FUNCTION_BLOCK FB_Escort_monitoring
VAR_INPUT
	Coil_Lh1:BOOL;
	Coil_Lh2:BOOL;
	Coil_Rh1:BOOL;
	Coil_Rh2:BOOL;
	Valve_Lh1_open:BOOL;
	Valve_Lh1_closed:BOOL;
	Valve_Lh2_open:BOOL;
	Valve_Lh2_closed:BOOL;
	Valve_Rh1_open:BOOL;
	Valve_Rh1_closed:BOOL;
	Valve_Rh2_open:BOOL;
	Valve_Rh2_closed:BOOL;
	Open_time:TIME;
	Close_time:TIME;
END_VAR
VAR_OUTPUT
	Lh1_not_opening:BOOL;
	Lh1_not_closing:BOOL;
	Lh1_open_and_closed:BOOL;
	Lh2_not_opening:BOOL;
	Lh2_not_closing:BOOL;
	Lh2_open_and_closed:BOOL;
	Rh1_not_opening:BOOL;
	Rh1_not_closing:BOOL;
	Rh1_open_and_closed:BOOL;
	Rh2_not_opening:BOOL;
	Rh2_not_closing:BOOL;
	Rh2_open_and_closed:BOOL;
	Lh1_with_brakes_on:BOOL;
	Lh2_with_brakes_on:BOOL;
	Rh1_with_brakes_on:BOOL;
	Rh2_with_brakes_on:BOOL;
	Lh1_Lh2_xcheck:BOOL;
	Rh1_Rh2_xcheck:BOOL;
	Lh1_chatter:BOOL;
	Lh2_chatter:BOOL;
	Rh1_chatter:BOOL;
	Rh2_chatter:BOOL;
END_VAR
VAR
	Reset_chatter_counters:BOOL;
	FB_Valve_monitor_0: FB_Valve_monitor;
	FB_Valve_monitor_1: FB_Valve_monitor;
	FB_Valve_monitor_2: FB_Valve_monitor;
	FB_Valve_monitor_3: FB_Valve_monitor;
	TON_0: TON;
	TON_1: TON;
	TON_2: TON;
	TON_3: TON;
	R_TRIG_0: R_TRIG;
	CTU_0: CTU;
	CTU_1: CTU;
	CTU_2: CTU;
	CTU_3: CTU;
END_VAR

Escort_valves();

METHOD Escort_valves
VAR_INPUT
END_VAR
{warning "TODO: Address %S7 needs to be correctly addressed}
VAR_INST // added by the converter: edge detectors and wires of the graphical bodies
    _w1, _w5 : ANY;
    _w2, _w3, _w4 : BOOL;
END_VAR
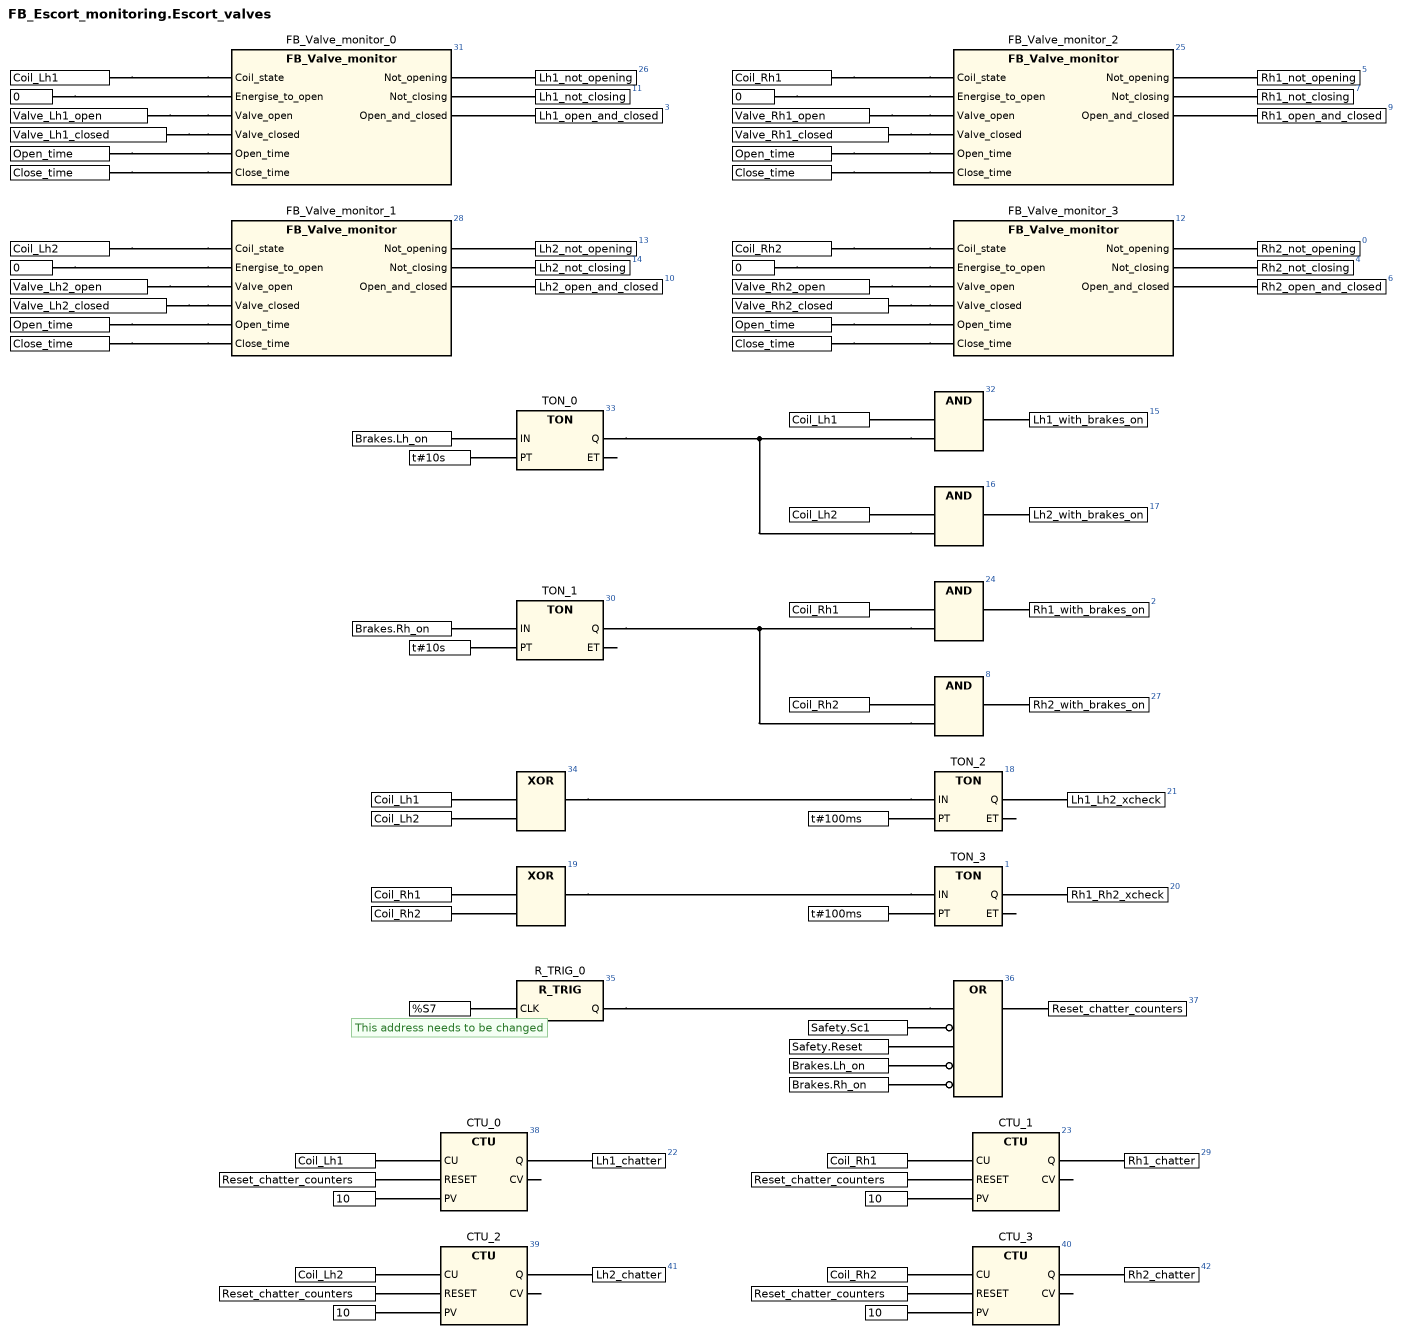
Rh2_not_opening := FB_Valve_monitor_3.Not_opening;
TON_3(IN := _w1, PT := t#100ms); // TON
Rh1_with_brakes_on := _w2;
Lh1_open_and_closed := FB_Valve_monitor_0.Open_and_closed;
Rh2_not_closing := FB_Valve_monitor_3.Not_closing;
Rh1_not_opening := FB_Valve_monitor_2.Not_opening;
Rh2_open_and_closed := FB_Valve_monitor_3.Open_and_closed;
Rh1_not_closing := FB_Valve_monitor_2.Not_closing;
_w3 := Coil_Rh2 AND TON_1.Q;
Rh1_open_and_closed := FB_Valve_monitor_2.Open_and_closed;
Lh2_open_and_closed := FB_Valve_monitor_1.Open_and_closed;
Lh1_not_closing := FB_Valve_monitor_0.Not_closing;
FB_Valve_monitor_3(
    Coil_state := Coil_Rh2,
    Energise_to_open := 0,
    Valve_open := Valve_Rh2_open,
    Valve_closed := Valve_Rh2_closed,
    Open_time := Open_time,
    Close_time := Close_time); // FB_Valve_monitor
Lh2_not_opening := FB_Valve_monitor_1.Not_opening;
Lh2_not_closing := FB_Valve_monitor_1.Not_closing;
Lh1_with_brakes_on := _w4;
Lh2_with_brakes_on := Coil_Lh2 AND TON_0.Q;
TON_2(IN := _w5, PT := t#100ms); // TON
_w1 := Coil_Rh1 XOR Coil_Rh2;
Rh1_Rh2_xcheck := TON_3.Q;
Lh1_Lh2_xcheck := TON_2.Q;
Lh1_chatter := CTU_0.Q;
CTU_1(CU := Coil_Rh1, RESET := Reset_chatter_counters, PV := 10); // CTU
_w2 := Coil_Rh1 AND TON_1.Q;
FB_Valve_monitor_2(
    Coil_state := Coil_Rh1,
    Energise_to_open := 0,
    Valve_open := Valve_Rh1_open,
    Valve_closed := Valve_Rh1_closed,
    Open_time := Open_time,
    Close_time := Close_time); // FB_Valve_monitor
Lh1_not_opening := FB_Valve_monitor_0.Not_opening;
Rh2_with_brakes_on := _w3;
FB_Valve_monitor_1(
    Coil_state := Coil_Lh2,
    Energise_to_open := 0,
    Valve_open := Valve_Lh2_open,
    Valve_closed := Valve_Lh2_closed,
    Open_time := Open_time,
    Close_time := Close_time); // FB_Valve_monitor
Rh1_chatter := CTU_1.Q;
TON_1(IN := Brakes.Rh_on, PT := t#10s); // TON
FB_Valve_monitor_0(
    Coil_state := Coil_Lh1,
    Energise_to_open := 0,
    Valve_open := Valve_Lh1_open,
    Valve_closed := Valve_Lh1_closed,
    Open_time := Open_time,
    Close_time := Close_time); // FB_Valve_monitor
_w4 := Coil_Lh1 AND TON_0.Q;
TON_0(IN := Brakes.Lh_on, PT := t#10s); // TON
_w5 := Coil_Lh1 XOR Coil_Lh2;
R_TRIG_0(CLK := %S7); // R_TRIG
Reset_chatter_counters := R_TRIG_0.Q OR NOT Safety.Sc1 OR Safety.Reset OR NOT Brakes.Lh_on OR NOT Brakes.Rh_on;
// This address needs to be changed
CTU_0(CU := Coil_Lh1, RESET := Reset_chatter_counters, PV := 10); // CTU
CTU_2(CU := Coil_Lh2, RESET := Reset_chatter_counters, PV := 10); // CTU
CTU_3(CU := Coil_Rh2, RESET := Reset_chatter_counters, PV := 10); // CTU
Lh2_chatter := CTU_2.Q;
Rh2_chatter := CTU_3.Q;
END_METHOD

END_FUNCTION_BLOCK

(* stored: Version 1.1.0.1, ProductVersion 3.1.4024.0
   POU FB_Escort_monitoring: Id {e0bab0e0-eb95-4538-8f03-d429982552ac}, SpecialFunc None
   Method Escort_valves: Id {d1d1eeab-a8ee-4c07-a484-13efd057e363} *)
